PROGRAM INTERNAL MAIN
VAR
    Context : MainContext;
END_VAR

END_PROGRAM

(* stored: Version 1.1.0.1, ProductVersion 3.1.4024.6
   POU MAIN: Id {0282f9e5-4698-05e8-2627-320dd5fad7b2}, SpecialFunc None *)
